{attribute 'Tc2GvlVarNames'}
VAR_GLOBAL CONSTANT
	(* AKM_Zustand_Regelung_Modus *)
	E_AKM_Regelung_Modus_T_KW					: SINT := -1;
	E_AKM_Regelung_Modus_T_WW					: SINT := 1;

	(* System_AKM_Zustand_Status *)
	E_System_AKM_Zustand_Status_Idle_Sperre		: SINT := 0;
	E_System_AKM_Zustand_Status_Betriebsbereit	: SINT := 1;
	E_System_AKM_Zustand_Status_Nachl			: SINT := 4;
	E_System_AKM_Zustand_Status_Vorl			: SINT := 5;
	E_System_AKM_Zustand_Status_Betrieb			: SINT := 8;
	E_System_AKM_Zustand_Status_Betrieb_Sperre	: SINT := 9;
	E_System_AKM_Zustand_Status_Stoerung		: SINT := 99;
END_VAR

(* stored: Version 1.1.0.1, ProductVersion 3.1.4024.9
   GVL Con_AKM: Id {a4ae4688-caa5-4fa6-8efb-da17aad47ff8} *)
